{attribute 'pack_mode' := '2'}
TYPE ST_AXIS_STATE :
STRUCT

  eState      : E_AXIS_STATE; // mirror the requested axis function; 
                                        // + E_PROGRESS
END_STRUCT
END_TYPE

(* stored: Version 1.1.0.1, ProductVersion 3.1.4024.12
   DUT ST_AXIS_STATE: Id {4769737f-c1e9-07b0-0307-e866a6addcfa} *)
